FUNCTION_BLOCK FB_digitalOut
VAR
	bOutput AT %Q* : BOOL;
END_VAR

METHOD turnOff : BOOL
VAR_INPUT
END_VAR
bOutput := FALSE;
END_METHOD

METHOD turnOn : BOOL
VAR_INPUT
END_VAR
bOutput := TRUE;
END_METHOD

END_FUNCTION_BLOCK

(* stored: Version 1.1.0.1, ProductVersion 3.1.4024.13
   POU FB_digitalOut: Id {9b8d181d-cfbc-4476-bcee-94eb362a3000}, SpecialFunc None
   Method turnOff: Id {4424f068-6486-4e26-9e95-7c1b3bbc0259}
   Method turnOn: Id {f53682b9-6e21-41f8-9c27-119a87670951} *)
